// TIA Portal V17 export
// export: Created 2025-06-20T10:18:00.170723Z, ExportSetting WithDefaults, DisplayName Totally Integrated Automation Portal, DisplayVersion V17 Update 8, DisplayName TIA Portal Openness, DisplayVersion V17 Update 8, DisplayName TIA Portal Version Control Interface, DisplayVersion V17, DisplayName SINAMICS Startdrive Advanced, DisplayVersion V17 SP2, DisplayName SINAMICS Startdrive G110M, G120, G120C, G120D, G120P, G115D, DisplayVersion V17 SP2, DisplayName SINAMICS Startdrive G130, G150, S120, S150, SINAMICS MV, S210, DisplayVersion V17 SP2, DisplayName STEP 7 Professional, DisplayVersion V17 Update 8, DisplayName SINUMERIK ONE STEP 7 Toolbox, DisplayVersion V17 Update 12, DisplayName SINUMERIK ONE PLC Basic Program Plus, DisplayVersion V17 Update 12, DisplayName SINUMERIK 840D sl STEP 7 Toolbox, DisplayVersion V17 Update 12, DisplayName STEP 7 Safety, DisplayVersion V17 Update 6, DisplayName WinCC Advanced, DisplayVersion V17 Update 8
FUNCTION_BLOCK "FB16001_METHODS_CONNECTION_MGR"   // FB16001, LAD
{ S7_Optimized_Access := 'FALSE' }
VERSION : 0.1
// stored: AutoNumber false, IsIECCheckEnabled false, SetENOAutomatically false, UDAEnableTagReadback false
   VAR_INPUT
      CONNECTION_BLOCK_DONE : Bool;   // DONE FROM CONNECTION BLOCK
      CONNECTION_BLOCK_ERROR : Bool;   // ERROR FROM CONNECTION BLOCK
      CONNECTION_BLOCK_BUSY : Bool;   // BUSY FROM CONNECT BLOCK
      READ_VARIABLES_BLOCK_ERROR : Bool;   // ERROR FROM READ VARIABLES BLOCK
      DISCONNECT_BLOCK_DONE : Bool;   // DONE FROM DISCONNECT BLOCK
      DISCONNECT_BLOCK_BUSY : Bool;   // BUSY FROM DISCONNECT BLOCK
      RESET_CONNECTION_ATTEMPTS : Bool;   // RESET CONNECTION ATTEMPTS
      OPC_UA_CONNECT_STATUS : DWord;   // OPC UA Connect Instance Status
      OPC_UA_GET_INDEX_LIST_STATUS : DWord;   // OPC UA GET INDEX LIST STATUS
      OPC_UA_GET_HANDLE_LIST_STATUS : DWord;   // OPC UA GE HANDLE LIST STATUS
      OPC_UA_GET_METHOD_LIST_STATUS : DWord;   // OPC UA GET METHOD HANLDE LIST STATUS
      OPC_UA_GET_METHOD_LIST_STATUS_1 : DWord;   // OPC UA GET METHOD HANLDE LIST STATUS
      OPC_UA_RELEASE_HANDLE_LIST_STATUS : DWord;   // OPC UA RELEASE HANDLE LIST STATUS
      OPC_UA_RELEASE_METHOD_LIST_STATUS : DWord;   // OPC UA RELEASE METHOD HANDLE LIST STATUS
      OPC_UA_RELEASE_METHOD_LIST_STATUS_1 : DWord;   // OPC UA RELEASE METHOD HANDLE LIST STATUS
      OPC_UA_READ_VARIABLES_STATUS : DWord;   // OPC UA READ VARIABLES STATUS
      OPC_UA_DISCONNECT_STATUS : DWord;   // OPC UA DISCONNECT STATUS
      OPC_UA_CONNECTION_GET_STATUS : DWord;   // OPC UA CONNECTION GET STATUS
      MAX_CON_ATTEMPTS : Int;   // MAX NUMBER OF CONNECTION ATTEMPTS
   END_VAR
   VAR_OUTPUT
      RETRY_CONNECTION : Bool;   // RETRY CONNECTION
      DISCONNECT : Bool;   // DISCONNECT
      CONNECTION_ERROR : Bool;   // CONNECTION ERROR
      CONNECTION_ERROR_STATUS : "CONNECTION_ERROR_STATUS";   // CONNECTION ERROR STATUS
   END_VAR
   VAR DB_SPECIFIC
      CONNECTION_ERROR_MEM : Bool;   // CONNECTION ERROR MEMORY
      CONNECTION_DONE_MEM : Bool;   // CONNECTION DONE MEMORY
      DISCONNECT_DONE_MEM : Bool;   // DISCONNECT DONE MEMORY
      ERROR_COUNTER : Int;   // CONNECTION ERROR COUNTER
      AUX_PULSE : Bool;   // AUX PULSE
      AUX_PULSE_1 : Bool;   // AUX PULSE 1
      AUX_PULSE_2 : Bool;   // AUX PULSE 2
      LAST_ERROR_TIME_STAMP : DTL;   // LAST ERROR TIME STAMP
      RET_VAL : Int;   // RET VAL
   END_VAR
   VAR_TEMP   // added for the SCL form of the ladder/FBD networks
      _w1 : Bool;
      _w2 : Bool;
   END_VAR
BEGIN

REGION Network 1: CONNECTION DONE INPUTS
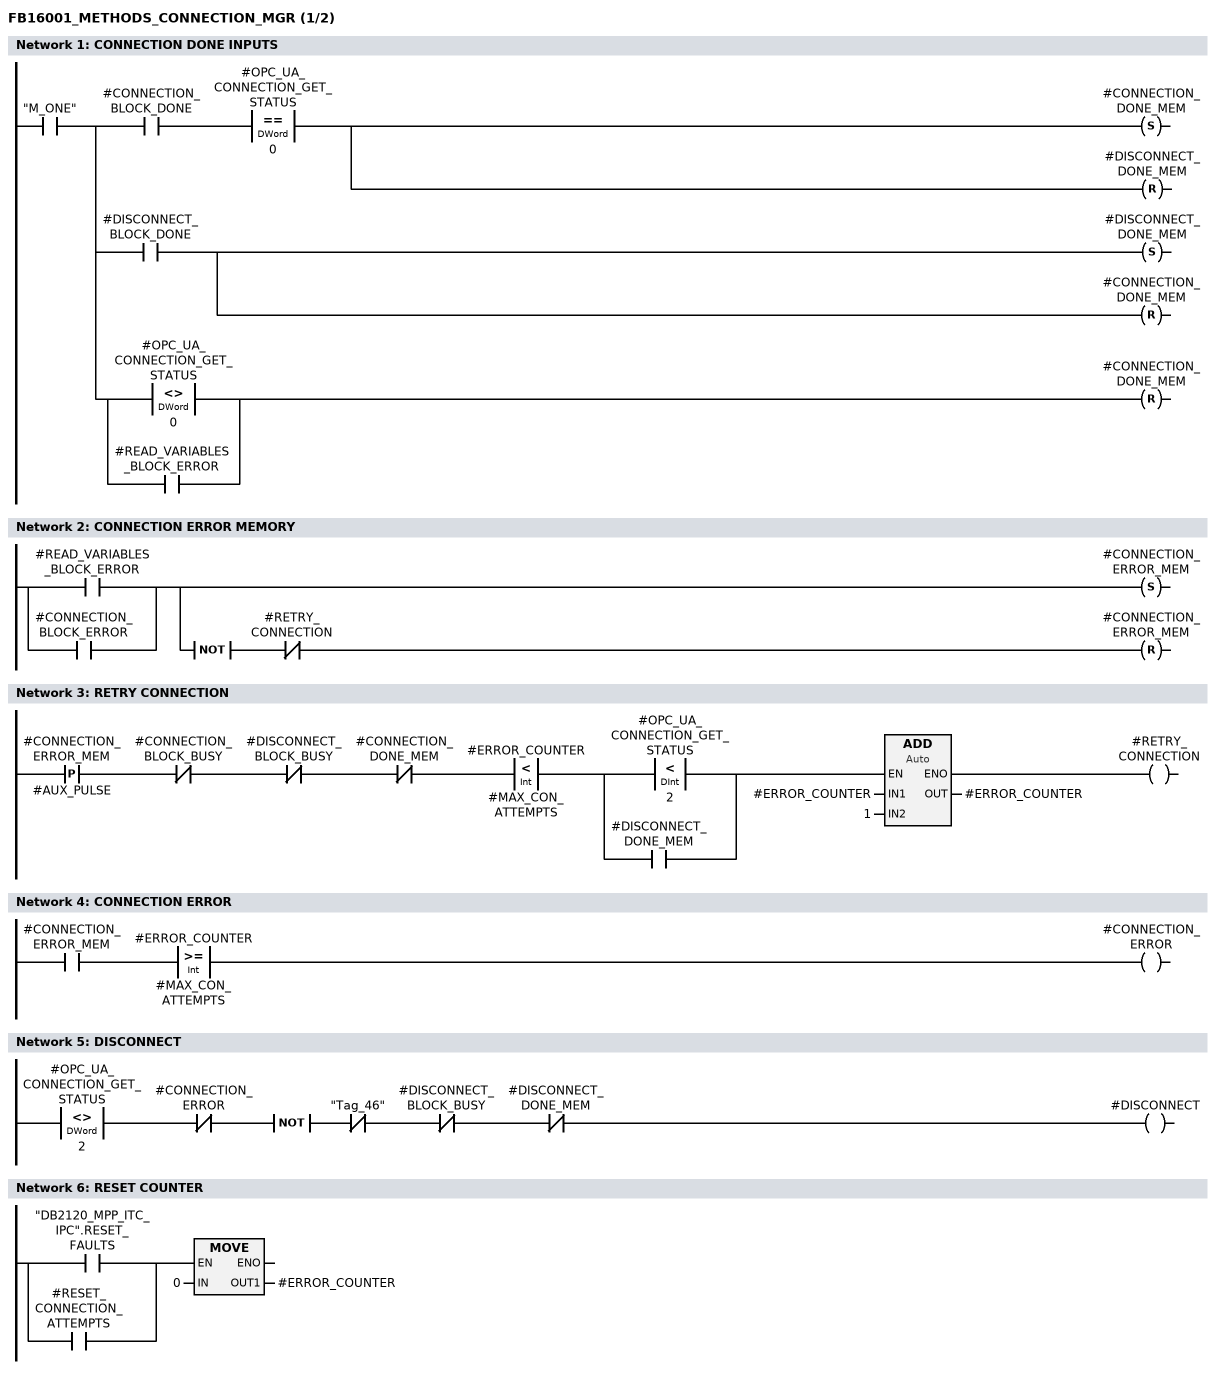
   RUNG wire#powerrail
      Contact( "M_ONE" )
      wire#w1
      Contact( #CONNECTION_BLOCK_DONE )
      { S7_Templates := "SrcType := DWord" } EQ_Contact(in1 := #OPC_UA_CONNECTION_GET_STATUS, in2 := 0)
      wire#w2
      S_Coil( #CONNECTION_DONE_MEM )
   END_RUNG
   RUNG wire#w2
      R_Coil( #DISCONNECT_DONE_MEM )
   END_RUNG
   RUNG wire#w1
      Contact( #DISCONNECT_BLOCK_DONE )
      wire#w3
      S_Coil( #DISCONNECT_DONE_MEM )
   END_RUNG
   RUNG wire#w3
      R_Coil( #CONNECTION_DONE_MEM )
   END_RUNG
   RUNG wire#w1
      { S7_Templates := "SrcType := DWord" } NE_Contact(in1 := #OPC_UA_CONNECTION_GET_STATUS, in2 := 0)
      wire#w4
      R_Coil( #CONNECTION_DONE_MEM )
   END_RUNG
   RUNG wire#w1
      Contact( #READ_VARIABLES_BLOCK_ERROR )
   END_RUNG wire#w4
   // the same network as SCL:
   IF "M_ONE" AND #CONNECTION_BLOCK_DONE AND (#OPC_UA_CONNECTION_GET_STATUS = 0) THEN
       #CONNECTION_DONE_MEM := TRUE;
       #DISCONNECT_DONE_MEM := FALSE;
   END_IF;
   IF "M_ONE" AND #DISCONNECT_BLOCK_DONE THEN
       #DISCONNECT_DONE_MEM := TRUE;
       #CONNECTION_DONE_MEM := FALSE;
   END_IF;
   IF "M_ONE" AND ((#OPC_UA_CONNECTION_GET_STATUS <> 0) OR #READ_VARIABLES_BLOCK_ERROR) THEN
       #CONNECTION_DONE_MEM := FALSE;
   END_IF;
END_REGION

REGION Network 2: CONNECTION ERROR MEMORY
   RUNG wire#powerrail
      Contact( #READ_VARIABLES_BLOCK_ERROR )
      wire#w1
      S_Coil( #CONNECTION_ERROR_MEM )
   END_RUNG
   RUNG wire#powerrail
      Contact( #CONNECTION_BLOCK_ERROR )
   END_RUNG wire#w1
   RUNG wire#w1
      Not()
      I_Contact( #RETRY_CONNECTION )
      R_Coil( #CONNECTION_ERROR_MEM )
   END_RUNG
   // the same network as SCL:
   #_w1 := #READ_VARIABLES_BLOCK_ERROR OR #CONNECTION_BLOCK_ERROR;
   IF #_w1 THEN #CONNECTION_ERROR_MEM := TRUE; END_IF;
   IF NOT #_w1 AND NOT #RETRY_CONNECTION THEN #CONNECTION_ERROR_MEM := FALSE; END_IF;
END_REGION

REGION Network 3: RETRY CONNECTION
   RUNG wire#powerrail
      P_Contact(operand := #CONNECTION_ERROR_MEM, bit := #AUX_PULSE)
      I_Contact( #CONNECTION_BLOCK_BUSY )
      I_Contact( #DISCONNECT_BLOCK_BUSY )
      I_Contact( #CONNECTION_DONE_MEM )
      { S7_Templates := "SrcType := Int" } LT_Contact(in1 := #ERROR_COUNTER, in2 := #MAX_CON_ATTEMPTS)
      wire#w1
      { S7_Templates := "SrcType := DInt" } LT_Contact(in1 := #OPC_UA_CONNECTION_GET_STATUS, in2 := 2)
      wire#w2
      Add(in1 := #ERROR_COUNTER, in2 := 1, out => #ERROR_COUNTER)
      Coil( #RETRY_CONNECTION )
   END_RUNG
   RUNG wire#w1
      Contact( #DISCONNECT_DONE_MEM )
   END_RUNG wire#w2
   // the same network as SCL:
   #_w1 := #CONNECTION_ERROR_MEM AND NOT #AUX_PULSE;   // rising edge of #CONNECTION_ERROR_MEM
   #AUX_PULSE := #CONNECTION_ERROR_MEM;
   #_w2 := #_w1 AND NOT #CONNECTION_BLOCK_BUSY AND NOT #DISCONNECT_BLOCK_BUSY AND NOT #CONNECTION_DONE_MEM AND (#ERROR_COUNTER < #MAX_CON_ATTEMPTS) AND ((#OPC_UA_CONNECTION_GET_STATUS < 2) OR #DISCONNECT_DONE_MEM);
   IF #_w2 THEN #ERROR_COUNTER := #ERROR_COUNTER + 1; END_IF;
   #RETRY_CONNECTION := #_w2;
END_REGION

REGION Network 4: CONNECTION ERROR
   RUNG wire#powerrail
      Contact( #CONNECTION_ERROR_MEM )
      { S7_Templates := "SrcType := Int" } GE_Contact(in1 := #ERROR_COUNTER, in2 := #MAX_CON_ATTEMPTS)
      Coil( #CONNECTION_ERROR )
   END_RUNG
   // the same network as SCL:
   #CONNECTION_ERROR := #CONNECTION_ERROR_MEM AND (#ERROR_COUNTER >= #MAX_CON_ATTEMPTS);
END_REGION

REGION Network 5: DISCONNECT
   RUNG wire#powerrail
      { S7_Templates := "SrcType := DWord" } NE_Contact(in1 := #OPC_UA_CONNECTION_GET_STATUS, in2 := 2)
      I_Contact( #CONNECTION_ERROR )
      Not()
      I_Contact( "Tag_46" )
      I_Contact( #DISCONNECT_BLOCK_BUSY )
      I_Contact( #DISCONNECT_DONE_MEM )
      Coil( #DISCONNECT )
   END_RUNG
   // the same network as SCL:
   #DISCONNECT := NOT ((#OPC_UA_CONNECTION_GET_STATUS <> 2) AND NOT #CONNECTION_ERROR) AND NOT "Tag_46" AND NOT #DISCONNECT_BLOCK_BUSY AND NOT #DISCONNECT_DONE_MEM;
END_REGION

REGION Network 6: RESET COUNTER
   RUNG wire#powerrail
      Contact( "DB2120_MPP_ITC_IPC".RESET_FAULTS )
      wire#w1
      Move(in := 0, out1 => #ERROR_COUNTER)
   END_RUNG
   RUNG wire#powerrail
      Contact( #RESET_CONNECTION_ATTEMPTS )
   END_RUNG wire#w1
   // the same network as SCL:
   IF "DB2120_MPP_ITC_IPC".RESET_FAULTS OR #RESET_CONNECTION_ATTEMPTS THEN #ERROR_COUNTER := 0; END_IF;
END_REGION

REGION Network 7: SAVE CONNECTION ERROR STATUS
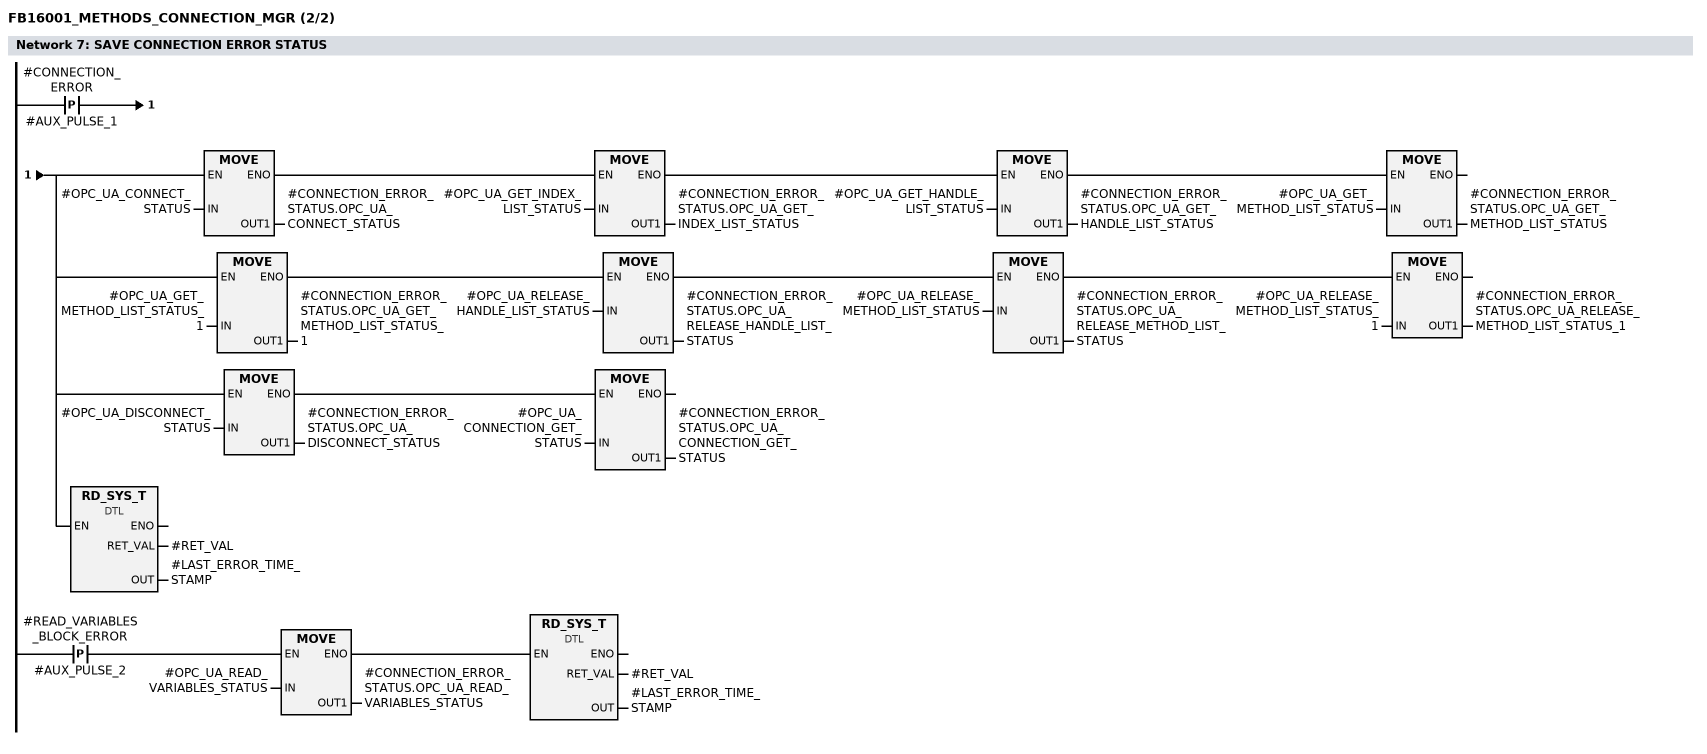
   RUNG wire#powerrail
      P_Contact(operand := #CONNECTION_ERROR, bit := #AUX_PULSE_1)
      wire#w1
      Move(in := #OPC_UA_CONNECT_STATUS, out1 => #CONNECTION_ERROR_STATUS.OPC_UA_CONNECT_STATUS)
      Move(in := #OPC_UA_GET_INDEX_LIST_STATUS, out1 => #CONNECTION_ERROR_STATUS.OPC_UA_GET_INDEX_LIST_STATUS)
      Move(in := #OPC_UA_GET_HANDLE_LIST_STATUS, out1 => #CONNECTION_ERROR_STATUS.OPC_UA_GET_HANDLE_LIST_STATUS)
      Move(in := #OPC_UA_GET_METHOD_LIST_STATUS, out1 => #CONNECTION_ERROR_STATUS.OPC_UA_GET_METHOD_LIST_STATUS)
   END_RUNG
   RUNG wire#w1
      Move(in := #OPC_UA_GET_METHOD_LIST_STATUS_1, out1 => #CONNECTION_ERROR_STATUS.OPC_UA_GET_METHOD_LIST_STATUS_1)
      Move(in := #OPC_UA_RELEASE_HANDLE_LIST_STATUS, out1 => #CONNECTION_ERROR_STATUS.OPC_UA_RELEASE_HANDLE_LIST_STATUS)
      Move(in := #OPC_UA_RELEASE_METHOD_LIST_STATUS, out1 => #CONNECTION_ERROR_STATUS.OPC_UA_RELEASE_METHOD_LIST_STATUS)
      Move(in := #OPC_UA_RELEASE_METHOD_LIST_STATUS_1, out1 => #CONNECTION_ERROR_STATUS.OPC_UA_RELEASE_METHOD_LIST_STATUS_1)
   END_RUNG
   RUNG wire#w1
      Move(in := #OPC_UA_DISCONNECT_STATUS, out1 => #CONNECTION_ERROR_STATUS.OPC_UA_DISCONNECT_STATUS)
      Move(in := #OPC_UA_CONNECTION_GET_STATUS, out1 => #CONNECTION_ERROR_STATUS.OPC_UA_CONNECTION_GET_STATUS)
   END_RUNG
   RUNG wire#w1
      { S7_Templates := "date_type := DTL" } RD_SYS_T(RET_VAL => #RET_VAL, OUT => #LAST_ERROR_TIME_STAMP)
   END_RUNG
   RUNG wire#powerrail
      P_Contact(operand := #READ_VARIABLES_BLOCK_ERROR, bit := #AUX_PULSE_2)
      Move(in := #OPC_UA_READ_VARIABLES_STATUS, out1 => #CONNECTION_ERROR_STATUS.OPC_UA_READ_VARIABLES_STATUS)
      { S7_Templates := "date_type := DTL" } RD_SYS_T(RET_VAL => #RET_VAL, OUT => #LAST_ERROR_TIME_STAMP)
   END_RUNG
   // the same network as SCL:
   #_w1 := #CONNECTION_ERROR AND NOT #AUX_PULSE_1;   // rising edge of #CONNECTION_ERROR
   #AUX_PULSE_1 := #CONNECTION_ERROR;
   IF #_w1 THEN
       #CONNECTION_ERROR_STATUS.OPC_UA_CONNECT_STATUS := #OPC_UA_CONNECT_STATUS;
       #CONNECTION_ERROR_STATUS.OPC_UA_GET_INDEX_LIST_STATUS := #OPC_UA_GET_INDEX_LIST_STATUS;
       #CONNECTION_ERROR_STATUS.OPC_UA_GET_HANDLE_LIST_STATUS := #OPC_UA_GET_HANDLE_LIST_STATUS;
       #CONNECTION_ERROR_STATUS.OPC_UA_GET_METHOD_LIST_STATUS := #OPC_UA_GET_METHOD_LIST_STATUS;
       #CONNECTION_ERROR_STATUS.OPC_UA_GET_METHOD_LIST_STATUS_1 := #OPC_UA_GET_METHOD_LIST_STATUS_1;
       #CONNECTION_ERROR_STATUS.OPC_UA_RELEASE_HANDLE_LIST_STATUS := #OPC_UA_RELEASE_HANDLE_LIST_STATUS;
       #CONNECTION_ERROR_STATUS.OPC_UA_RELEASE_METHOD_LIST_STATUS := #OPC_UA_RELEASE_METHOD_LIST_STATUS;
       #CONNECTION_ERROR_STATUS.OPC_UA_RELEASE_METHOD_LIST_STATUS_1 := #OPC_UA_RELEASE_METHOD_LIST_STATUS_1;
       #CONNECTION_ERROR_STATUS.OPC_UA_DISCONNECT_STATUS := #OPC_UA_DISCONNECT_STATUS;
       #CONNECTION_ERROR_STATUS.OPC_UA_CONNECTION_GET_STATUS := #OPC_UA_CONNECTION_GET_STATUS;
       #RET_VAL := RD_SYS_T(OUT => #LAST_ERROR_TIME_STAMP);
   END_IF;
   #_w2 := #READ_VARIABLES_BLOCK_ERROR AND NOT #AUX_PULSE_2;   // rising edge of #READ_VARIABLES_BLOCK_ERROR
   #AUX_PULSE_2 := #READ_VARIABLES_BLOCK_ERROR;
   IF #_w2 THEN
       #CONNECTION_ERROR_STATUS.OPC_UA_READ_VARIABLES_STATUS := #OPC_UA_READ_VARIABLES_STATUS;
       #RET_VAL := RD_SYS_T(OUT => #LAST_ERROR_TIME_STAMP);
   END_IF;
END_REGION
END_FUNCTION_BLOCK
